FUNCTION_BLOCK FB_SysLogExporter IMPLEMENTS I_Visitor
VAR_INPUT
END_VAR
VAR_OUTPUT
END_VAR
VAR
END_VAR

METHOD visitConveyor
VAR_INPUT
	fbConveyor : FB_Conveyor;
END_VAR
ADSLOGSTR( msgCtrlMask := ADSLOG_MSGTYPE_LOG, msgFmtStr := '', strArg := '');
ADSLOGSTR( msgCtrlMask := ADSLOG_MSGTYPE_LOG, msgFmtStr := 'PLC Msg. *** Printing Messages For: %s', strArg := fbConveyor.pPath);
ADSLOGSTR( msgCtrlMask := ADSLOG_MSGTYPE_LOG, msgFmtStr := CONCAT(fbConveyor.pPath,':: Status := %s'), strArg := TO_STRING(fbConveyor.pStatus));
ADSLOGSTR( msgCtrlMask := ADSLOG_MSGTYPE_LOG, msgFmtStr := CONCAT(fbConveyor.pPath,':: Velocity := %s'), strArg := TO_STRING(fbConveyor.pVelocity));
ADSLOGSTR( msgCtrlMask := ADSLOG_MSGTYPE_LOG, msgFmtStr := CONCAT(fbConveyor.pPath,':: Position := %s'), strArg := TO_STRING(fbConveyor.pPosition));
END_METHOD

METHOD visitHeater
VAR_INPUT
	fbHeater : FB_Heater;
END_VAR
ADSLOGSTR( msgCtrlMask := ADSLOG_MSGTYPE_LOG, msgFmtStr := '', strArg := '');
ADSLOGSTR( msgCtrlMask := ADSLOG_MSGTYPE_LOG, msgFmtStr := 'PLC Msg. *** Printing Messages For: %s', strArg := fbHeater.pPath);
ADSLOGSTR( msgCtrlMask := ADSLOG_MSGTYPE_LOG, msgFmtStr := CONCAT(fbHeater.pPath,':: Status := %s'), strArg := TO_STRING(fbHeater.pStatus));
ADSLOGSTR( msgCtrlMask := ADSLOG_MSGTYPE_LOG, msgFmtStr := CONCAT(fbHeater.pPath,':: Temperature := %s'), strArg := TO_STRING(fbHeater.pTemp));
END_METHOD

METHOD visitIPC
VAR_INPUT
	fbIPC : FB_IPCDiagnostics;
END_VAR
ADSLOGSTR( msgCtrlMask := ADSLOG_MSGTYPE_LOG, msgFmtStr := '', strArg := '');
ADSLOGSTR( msgCtrlMask := ADSLOG_MSGTYPE_LOG, msgFmtStr := 'PLC Msg. *** Printing Messages For: %s', strArg := fbIPC.pPath);
ADSLOGSTR( msgCtrlMask := ADSLOG_MSGTYPE_LOG, msgFmtStr := CONCAT(fbIPC.pPath,':: CPU Usage := %s'), strArg := TO_STRING(fbIPC.pCPU_Usage));
ADSLOGSTR( msgCtrlMask := ADSLOG_MSGTYPE_LOG, msgFmtStr := CONCAT(fbIPC.pPath,':: CPU Temperature (F) := %s'), strArg := TO_STRING(fbIPC.pCPU_Temp));
END_METHOD

END_FUNCTION_BLOCK

(* stored: Version 1.1.0.1, ProductVersion 3.1.4024.12
   POU FB_SysLogExporter: Id {0dee553f-9ccd-492f-99ce-bf5953c98bd3}, SpecialFunc None
   Method visitConveyor: Id {0484067d-9c5e-4b40-ab70-934765cdac38}
   Method visitHeater: Id {eb907004-7ed4-41c6-95f0-edd3c6e91274}
   Method visitIPC: Id {b9910925-b6f1-49cd-8635-32e88c1bc861} *)
